INTERFACE I_LocalSystemTimeProvider

METHOD PUBLIC ConvertToString : I_DateTimeToStringConverter
VAR_INPUT
END_VAR
END_METHOD

{attribute 'monitoring':='variable'}
// Gets current system timo info as a <ST_CurrentSystemTimeInfo>
PROPERTY CurrentTime : REFERENCE TO ST_CurrentSystemTimeInfo
GET
END_GET
END_PROPERTY

END_INTERFACE

(* stored: Version 1.1.0.1, ProductVersion 3.1.4024.14
   Itf I_LocalSystemTimeProvider: Id {739de1b2-7958-07bc-150b-17ae5e4fc476}
   Method ConvertToString: Id {44adc15c-19ac-0a67-2299-2e503992cd1d}
   Property CurrentTime: Id {dc69b815-82ab-011b-2f1d-6f6ae8497b56}
   Get Get: Id {e71af7c8-9bcc-0614-14bc-beaaca577c88} *)
